Fanuc KAREL source: V_FIND_VLINE.kl

PROGRAM T
%NOLOCKGROUP
VAR
 v0 : STRING[40]
 v1 : INTEGER
 v2 : INTEGER
 v3 : PATH
 v4 : INTEGER
BEGIN
 V_FIND_VLINE(v0, v1, v2, v3, v4)
END T
